// TIA Portal V19 export
TYPE "LEXCHANGETRAY_typeSr1000ProfinetTelegram_userData128Byte"
// stored: Access Published
   STRUCT
      dataBytes : Array[0..127] of Byte;
      userDataSize : UInt;
      userData0 : Char;
      userData1 : Char;
      userData2 : Char;
      userData3 : Char;
      userData4 : Char;
      userData5 : Char;
      userData6 : Char;
      userData7 : Char;
      userData8 : Char;
      userData9 : Char;
      userData10 : Char;
      userData11 : Char;
      userData12 : Char;
      userData13 : Char;
      userData14 : Char;
      userData15 : Char;
   END_STRUCT;
END_TYPE
